FUNCTION SCALE_REAL_TO_UDINT : UDINT
VAR_INPUT
	I : REAL;
	Range_LL : REAL;
	Range_UL : REAL;
END_VAR
VAR
END_VAR

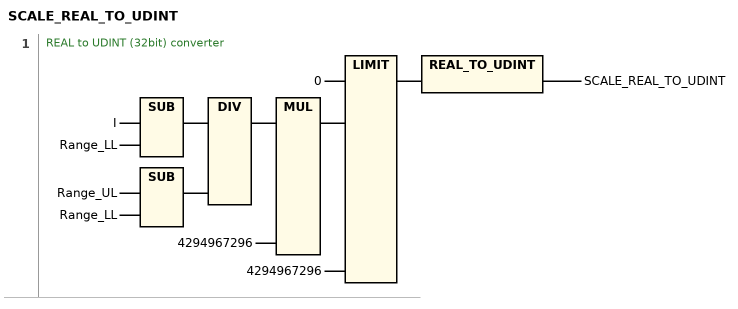
// NETWORK 1
// REAL to UDINT (32bit) converter
SCALE_REAL_TO_UDINT := REAL_TO_UDINT(LIMIT(0, ((I - Range_LL) / (Range_UL - Range_LL)) * 4294967296, 4294967296));

END_FUNCTION

(* stored: Version 1.1.0.1, ProductVersion 3.1.4024.6
   POU SCALE_REAL_TO_UDINT: Id {7dec20d6-90a6-4a61-9163-e8335c948398}, SpecialFunc None *)
